{attribute 'linkalways'} 
{attribute 'no_explicit_call' := 'This FB is a CLASS and must be accessed using methods or properties'}
{attribute 'enable_dynamic_creation'}
FUNCTION_BLOCK _TcVnVector2_REAL EXTENDS AliasDatatypeBase
VAR
	localData : TcVnVector2_REAL;
	activeData : REFERENCE TO TcVnVector2_REAL REF= localData;
	aliasBaseDatatype : _Array0to1OfREAL;
END_VAR

PROPERTY PUBLIC Address : PVOID
GET
Address := ADR(activeData);
END_GET
END_PROPERTY

METHOD PUBLIC ClearReference
VAR_INPUT
END_VAR
activeData REF= localData;
SetBaseDatatypeReference();
END_METHOD

METHOD PUBLIC Clone : I_Datatype
VAR
    pClone : POINTER TO _TcVnVector2_REAL;
END_VAR
pClone := __NEW(_TcVnVector2_REAL);
Clone := pClone^;
END_METHOD

METHOD FB_init : BOOL
VAR_INPUT
	bInitRetains : BOOL; // if TRUE, the retain variables are initialized (warm start / cold start)
	bInCopyCode : BOOL;  // if TRUE, the instance afterwards gets moved into the copy code (online change)
	//InitialValue : <type>; // if possible, not all values can be initialized
END_VAR
//localData := InitialValue; // if possible, not all values can be initialized
SetBaseDatatypeReference();
AddBaseDatatype(aliasBaseDatatype);
END_METHOD

PROPERTY PUBLIC Identifier : T_MAXSTRING
GET
Identifier := 'TcVnVector2_REAL';
END_GET
END_PROPERTY

METHOD PUBLIC MakeReferenceTo
VAR_INPUT
	ReferenceTarget : REFERENCE TO TcVnVector2_REAL;
END_VAR
activeData REF= ReferenceTarget;
SetBaseDatatypeReference();
END_METHOD

METHOD PROTECTED SetBaseDatatypeReference
VAR_INPUT
END_VAR
aliasBaseDatatype.MakeReferenceTo(activeData);
END_METHOD

PROPERTY PUBLIC Size : UDINT
GET
Size := SIZEOF(activeData);
END_GET
END_PROPERTY

METHOD TryMakeReferenceTo : BOOL
VAR_INPUT
	Target : I_Datatype;
END_VAR
VAR
	targetAsAlias : I_AliasDatatype;
	pTargetData : POINTER TO TcVnVector2_REAL;
END_VAR
IF NOT Target.TryResolveAsAliasDatatype(targetAsAlias) THEN
	RETURN;
END_IF

IF targetAsAlias.Identifier <> Identifier THEN
	RETURN;
END_IF

pTargetData := Target.Address;
activeData REF= pTargetData^;
SetBaseDatatypeReference();
TryMakeReferenceTo := TRUE;
END_METHOD

PROPERTY PUBLIC Value : REFERENCE TO TcVnVector2_REAL
GET
Value REF= activeData;
END_GET
END_PROPERTY

END_FUNCTION_BLOCK

(* stored: Version 1.1.0.1, ProductVersion 3.1.4024.13
   POU _TcVnVector2_REAL: Id {1d8df769-f7f2-0a0e-1951-d8c547dd805b}, SpecialFunc None
   Folder Core: Id {ed79e6d0-c65c-07ab-3a29-cce25b1b18c9}
   Folder Protected: Id {e8481c36-14b6-0a11-216a-a50ed8473cf2}
   Folder Customize: Id {02a20089-ac9f-093e-261d-f03a2f8f07cd}
   Folder Constructor: Id {05b193d1-0497-0cda-293c-79d7aeba4824}
   Property Address: Id {0f0cb079-cb2a-046e-1b7f-f6b095d070ea}
   Get Get: Id {8f26e8ed-fcdf-0c93-093b-0d134f5078a9}
   Method ClearReference: Id {08365816-2632-0670-1fe2-5580335c9877}
   Method Clone: Id {6a5ab1b6-187e-03a7-18ef-828e7478fcc3}
   Method FB_init: Id {be28e8b9-70f6-064e-134e-d943aa209bf8}
   Property Identifier: Id {c8adec2d-7b38-0e51-1c6f-c5b4ec75a1e0}
   Get Get: Id {038c2128-096e-0b65-213a-77b42d87808d}
   Method MakeReferenceTo: Id {a9374979-350e-0163-3f3a-f43d50e14864}
   Method SetBaseDatatypeReference: Id {8ef9c731-c7f4-05ac-3c1a-5a55b896c25b}
   Property Size: Id {f7598da6-c890-05ca-0f43-077b8a547424}
   Get Get: Id {f3ed89b1-f5d9-0f46-2539-d07be7098f9c}
   Method TryMakeReferenceTo: Id {f56696f3-afc0-0b87-1ccf-672ad37133f8}
   Property Value: Id {87bcf902-75af-0e53-334a-c1d4b2ef9fca}
   Get Get: Id {7f2b2c29-b732-074c-2c4a-646d5ca20607} *)
